// TIA Portal V17 export
// export: Created 2021-12-03T08:12:53.0003806Z, ExportSetting WithDefaults, DisplayName Totally Integrated Automation Portal, DisplayVersion V17, DisplayName TIA Portal Openness, DisplayVersion V17, DisplayName TIA Portal Version Control Interface, DisplayVersion V17, DisplayName STEP 7 Professional, DisplayVersion V17, DisplayName STEP 7 Safety, DisplayVersion V17, DisplayName WinCC Advanced, DisplayVersion V17
DATA_BLOCK "GDB_PlcToHmi"   // DB1000
VERSION : 0.1
// stored: AutoNumber false, IsOnlyStoredInLoadMemory false, IsWriteProtectedInAS false
   VAR
      Status : Struct
         EmrStp : Struct
            P1 : Int;   // Пульт P1
            P2 : Int;   // Пульт P2
            P3 : Int;   // Пульт P3
            Acc : Int;   // Ускоритель
            AccConsole : Int;   // Консоль ускорителя
            Dosim : Int;   // Дозиметр
            Gen : Int;   // Общий аварийный останов
         END_STRUCT;
         FrqConv : Struct
            ActSpeed : Int;   // Текщая скорость
            ActCurrent : Real;   // Текущий ток
            ActFault : Int;   // Текущая ошибка
            RefSpeed : Int;   // Запрашиваемая скорость
         END_STRUCT;
         Pwr : Int;   // Питание
         Sft : Int;   // Безопасность
         Acc : Int;   // Ускоритель
         Pwr_All : Int;   // Питание всех устройств
         BrkCirc : Int;   // Состояние автоматических выключателей
         Cmd : Int;   // Состояние вспомогательных команд
         Mod400_RlyOn : Int;   // Модулятор 400
         Mod230_RlyOn : Int;   // Модулятор 230
         Chill_RlyOn : Int;   // Чиллер
         Acc_RlyOn : Int;   // Ускоритель
         Conv_RlyOn : Int;   // Конвейер
         ConvActState : Int;   // Состояние конвейера
         ConvSns : Int;   // Состояние фотоэлектрических датчиков конвейера
         ChilPwrOffDlyTm : Time;   // Время отключения чиллера
         ChilPwrOnDlyTm : Time;   // Время включения чиллера
         AccCs_StateNr : Int;   // Состояние ускорителя
         ScanSeq_Sts : Int;   // Состояние последовательности сканирования
         FactSpeedCalc : Int;   // Фактическая скорость расчетная
         DetLine_Sts : Int;   // Статус детекторной линейки
         DetLine_TrigRate : Int;   // Частота детекторной линейки
         DetLine_ErgMode : Int;   // Режим энергии
         Animation : Int;   // Анимация кубика
      END_STRUCT;
      Faults : Struct
         FeedBack : Struct
            "24V" : Int;
            "220V" : Int;
            "380V" : Int;
            Control : Int;
         END_STRUCT;
         EmStBt : Int;
         Conveyer : Int;
      END_STRUCT;
   END_VAR
BEGIN
END_DATA_BLOCK
